// TIA Portal V18 export
VAR_GLOBAL   // PLC tag table "Variablentabelle_1"
   "a" AT %I0.0 : Bool;
   "b#" AT %I0.1 : Bool;
   c AT %I0.2 : Bool;
END_VAR
